FUNCTION_BLOCK SGReadyHeatPumpAdapter (* Actor for sending data to the SG Ready Heat Pump Adapter plugin controller in Polysun. *)
  (* Standard: 61499-2 *)
  (* Version 1.0, 2017-07-21, Marc Jakobi, HTW Berlin *)
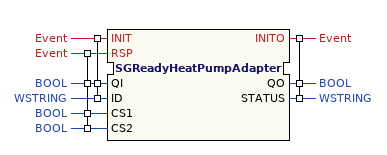
  EVENT_INPUT
    INIT WITH QI, ID; (* Service Initialization *)
    RSP WITH CS1, QI, CS2; (* Service Response *)
  END_EVENT
  EVENT_OUTPUT
    INITO WITH QO, STATUS; (* Initialization Confirm *)
  END_EVENT
  VAR_INPUT
    QI : BOOL; (* Input event qualifier *)
    ID : WSTRING; (* Connection Identifier *)
    CS1 : BOOL; (* SG-Ready control signal 1 *)
    CS2 : BOOL; (* SG-Ready control signal 2 *)
  END_VAR
  VAR_OUTPUT
    QO : BOOL; (* Output event qualifier *)
    STATUS : WSTRING; (* Service status *)
  END_VAR
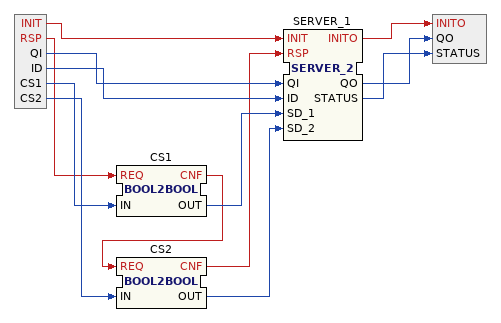
  FBS
    SERVER_1 : SERVER_2;
    CS1 : BOOL2BOOL;
    CS2 : BOOL2BOOL;
  END_FBS
  EVENT_CONNECTIONS
    INIT TO SERVER_1.INIT;
    SERVER_1.INITO TO INITO;
    RSP TO CS1.REQ;
    CS1.CNF TO CS2.REQ;
    CS2.CNF TO SERVER_1.RSP;
  END_CONNECTIONS
  DATA_CONNECTIONS
    QI TO SERVER_1.QI;
    ID TO SERVER_1.ID;
    SERVER_1.QO TO QO;
    SERVER_1.STATUS TO STATUS;
    CS1 TO CS1.IN;
    CS2 TO CS2.IN;
    CS1.OUT TO SERVER_1.SD_1;
    CS2.OUT TO SERVER_1.SD_2;
  END_CONNECTIONS
END_FUNCTION_BLOCK
